// Implicitly generated code : DO NOT EDIT
FUNCTION CheckDivDInt : DINT
VAR_INPUT
	divisor:DINT;
END_VAR

// Implicitly generated code : Only an Implementation suggestion
{noflow}
Fault_Count_G(CU:=FALSE) ; 
IF divisor = 0 THEN
	CheckDivDInt:=1;
		Fault_Count_G(CU:=TRUE) ; 
ELSE
	CheckDivDInt:=divisor;
END_IF;
{flow}

END_FUNCTION

(* stored: Version 1.1.0.1, ProductVersion 3.1.4024.2
   POU CheckDivDInt: Id {d6bc86ed-2140-44c0-9794-b7078c147bb0}, SpecialFunc CheckDivInt32 *)
